// TIA Portal V19 export
TYPE "LAF_typeMemCardMessages"
TITLE = SiemensMemoryCard diagnostic messages / SiemensMemoryCard DIagnsoe Meldungen
// Type contains the possible messages generated by the SMCDiag function. / SMC Diagnose Meldungen
// stored: Access Published
   STRUCT
      invalidValueModeParam { ExternalAccessible := 'False'; ExternalVisible := 'False'; ExternalWritable := 'False'} : Bool;   // 8080 Ungültiger Wert des Parameters "Mode" / 8080 Invalid value of the "Mode" parameter
      noMemCardInserted { ExternalAccessible := 'False'; ExternalVisible := 'False'; ExternalWritable := 'False'} : Bool;   // 8081 Keine SIMATIC Memory Card gesteckt (nur S7-1200) / 8081 No SIMATIC memory card inserted
      noDataAvailable { ExternalAccessible := 'False'; ExternalVisible := 'False'; ExternalWritable := 'False'} : Bool;   // 8092 Keine Daten verfügbar, z. B. weil "GetSMCinfo" von der CPU/SMC nicht unterstützt wird / 8092 No data available, for example, because "GetSMCinfo" is not supported by the PLC/SMC
      maxCallsReached { ExternalAccessible := 'False'; ExternalVisible := 'False'; ExternalWritable := 'False'} : Bool;   // 80C3 Die maximale Anzahl gleichzeitiger Aufrufe der Anweisung "GetSMCinfo" ist zur Zeit erreicht / 80C3 The maximum number of simultaneous calls of the "GetSMCinfo" instruction has been reached
      configMemSpaceWarning { ExternalAccessible := 'False'; ExternalVisible := 'False'; ExternalWritable := 'False'} : Bool;   // Parametrierte Speicherkapazität-Warnung erreicht / Parametrized Memory Space Warning reached
      configMemSpaceAlarm { ExternalAccessible := 'False'; ExternalVisible := 'False'; ExternalWritable := 'False'} : Bool;   // Parametrierte Speicherkapazität-Alarm erreicht / Parametrized Memory Space Alarm reached
      usedLiftetimeInvalid { ExternalAccessible := 'False'; ExternalVisible := 'False'; ExternalWritable := 'False'} : Bool;   // Verbrauchter Anteil Lebensdauer größer Parametrierter Anteil Lebensdauer / Used Lifetime bigger than parametrized Lifetime
      diagAlarmDisabled { ExternalAccessible := 'False'; ExternalVisible := 'False'; ExternalWritable := 'False'} : Bool;   // S7-1500 & S7-PLCSIM oder Diagnosealarm gesperrt (CPU Eigenschaften > SIMATIC Memory Card) / S7-1500 & S7-PLCSIM or diagnostic alarm disabled (PLC properties > SIMATIC Memory Card)
   END_STRUCT;
END_TYPE
